{attribute 'GeneratedUsingTerminal: EJ5101-0000-0016'}
{attribute addProperty BoxType "EJ5101-0000-0016"}
{attribute addProperty Id "StatusAT %I*Status_D8D782C316Counter_valueAT %I*UINT2Latch_valueAT %I*UINT2"}
{attribute addProperty CRC "2100585715"}
{attribute addProperty Size "20"}
TYPE ENC_Status_compact_7D3464F3 EXTENDS InputBase_8311D824 :
STRUCT
	{attribute addProperty Name "Status"}
	Status AT %I* : Status_D8D782C3;
	{attribute addProperty Name "Counter_value"}
	Counter_value AT %I* : UINT;
	{attribute addProperty Name "Latch_value"}
	Latch_value AT %I* : UINT;
END_STRUCT
END_TYPE
